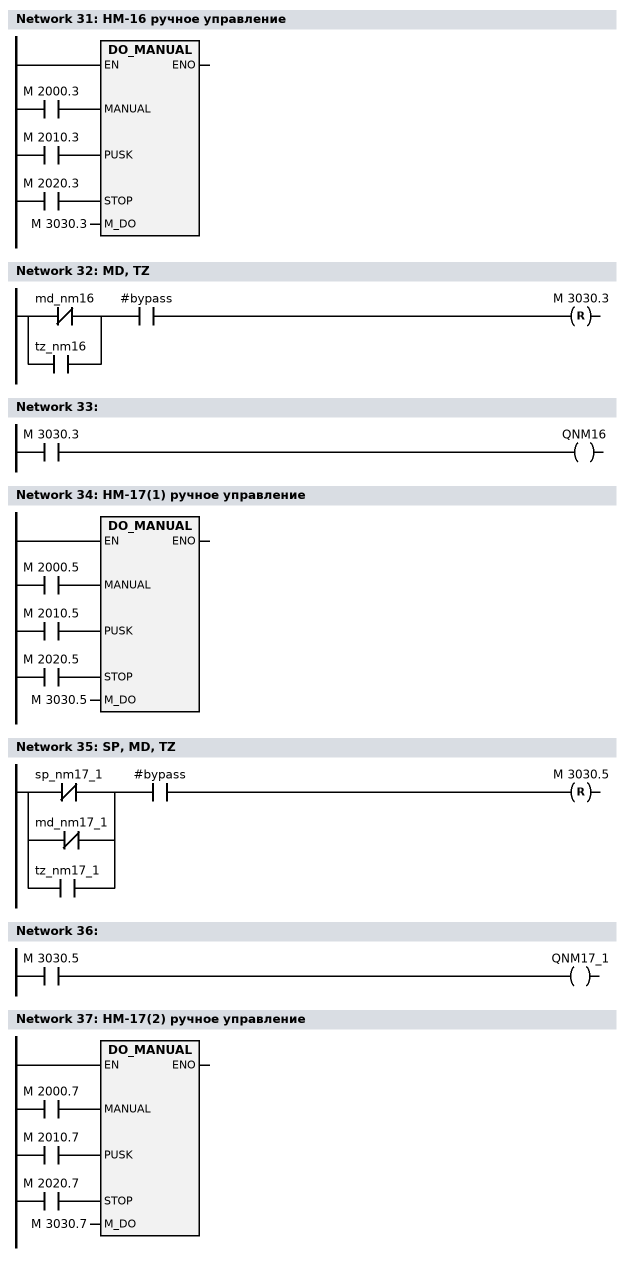
[picture p24: OB 1 networks 31-37]
NETWORK
TITLE = НМ-16 ручное управление
      A     M 2000.3;
      =     L 38.0;
      BLD   103;
      A     M 2010.3;
      =     L 38.1;
      BLD   103;
      A     M 2020.3;
      =     L 38.2;
      BLD   103;
      CALL  "DO_MANUAL" (
           MANUAL                   := L 38.0,
           PUSK                     := L 38.1,
           STOP                     := L 38.2,
           M_DO                     := M 3030.3);
      NOP   0;
NETWORK
TITLE = MD, TZ 
      A(;
      ON    "md_nm16";
      O     "tz_nm16";
      );
      A     #bypass;
      R     M 3030.3;
NETWORK
TITLE =
      A     M 3030.3;
      =     "QNM16";
NETWORK
TITLE = НМ-17(1) ручное управление
      A     M 2000.5;
      =     L 38.0;
      BLD   103;
      A     M 2010.5;
      =     L 38.1;
      BLD   103;
      A     M 2020.5;
      =     L 38.2;
      BLD   103;
      CALL  "DO_MANUAL" (
           MANUAL                   := L 38.0,
           PUSK                     := L 38.1,
           STOP                     := L 38.2,
           M_DO                     := M 3030.5);
      NOP   0;
NETWORK
TITLE = SP, MD, TZ 
      A(;
      ON    "sp_nm17_1";
      ON    "md_nm17_1";
      O     "tz_nm17_1";
      );
      A     #bypass;
      R     M 3030.5;
NETWORK
TITLE =
      A     M 3030.5;
      =     "QNM17_1";
NETWORK
TITLE = НМ-17(2) ручное управление
      A     M 2000.7;
      =     L 38.0;
      BLD   103;
      A     M 2010.7;
      =     L 38.1;
      BLD   103;
      A     M 2020.7;
      =     L 38.2;
      BLD   103;
      CALL  "DO_MANUAL" (
           MANUAL                   := L 38.0,
           PUSK                     := L 38.1,
           STOP                     := L 38.2,
           M_DO                     := M 3030.7);
      NOP   0;
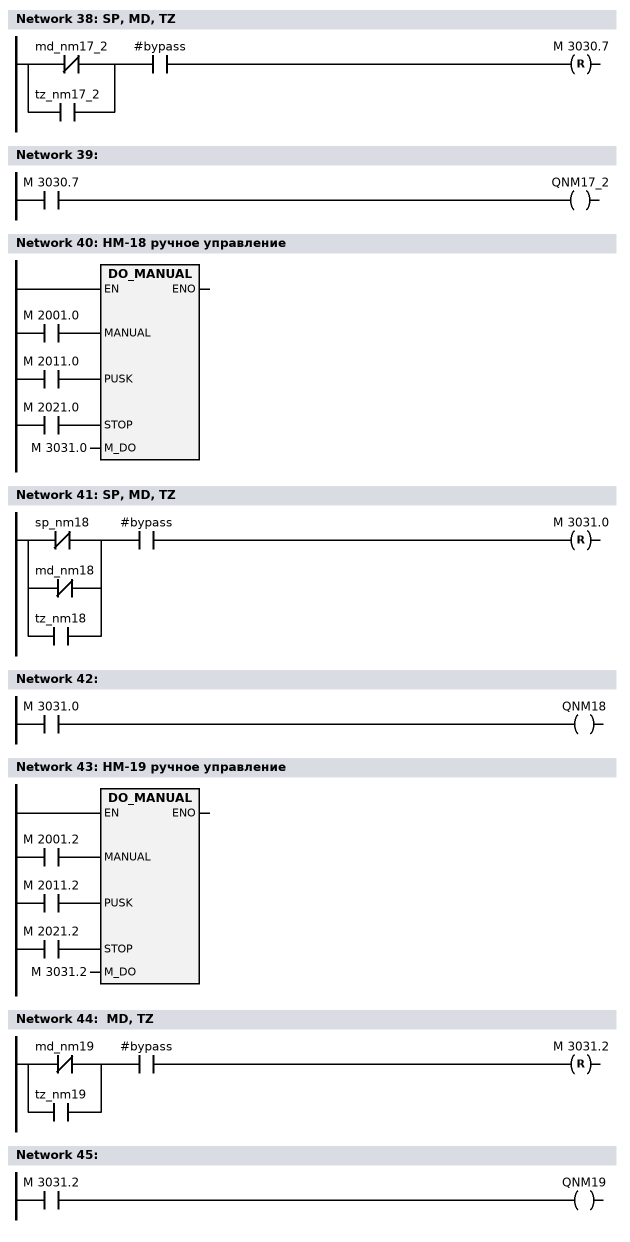
NETWORK
TITLE = SP, MD, TZ 
      A(;
      ON    "md_nm17_2";
      O     "tz_nm17_2";
      );
      A     #bypass;
      R     M 3030.7;
NETWORK
TITLE =
      A     M 3030.7;
      =     "QNM17_2";
NETWORK
TITLE = НМ-18 ручное управление
      A     M 2001.0;
      =     L 38.0;
      BLD   103;
      A     M 2011.0;
      =     L 38.1;
      BLD   103;
      A     M 2021.0;
      =     L 38.2;
      BLD   103;
      CALL  "DO_MANUAL" (
           MANUAL                   := L 38.0,
           PUSK                     := L 38.1,
           STOP                     := L 38.2,
           M_DO                     := M 3031.0);
      NOP   0;
NETWORK
TITLE = SP, MD, TZ 
      A(;
      ON    "sp_nm18";
      ON    "md_nm18";
      O     "tz_nm18";
      );
      A     #bypass;
      R     M 3031.0;
NETWORK
TITLE =
      A     M 3031.0;
      =     "QNM18";
NETWORK
TITLE = НМ-19 ручное управление
      A     M 2001.2;
      =     L 38.0;
      BLD   103;
      A     M 2011.2;
      =     L 38.1;
      BLD   103;
      A     M 2021.2;
      =     L 38.2;
      BLD   103;
      CALL  "DO_MANUAL" (
           MANUAL                   := L 38.0,
           PUSK                     := L 38.1,
           STOP                     := L 38.2,
           M_DO                     := M 3031.2);
      NOP   0;
NETWORK
TITLE =  MD, TZ 
      A(;
      ON    "md_nm19";
      O     "tz_nm19";
      );
      A     #bypass;
      R     M 3031.2;
NETWORK
TITLE =
      A     M 3031.2;
      =     "QNM19";
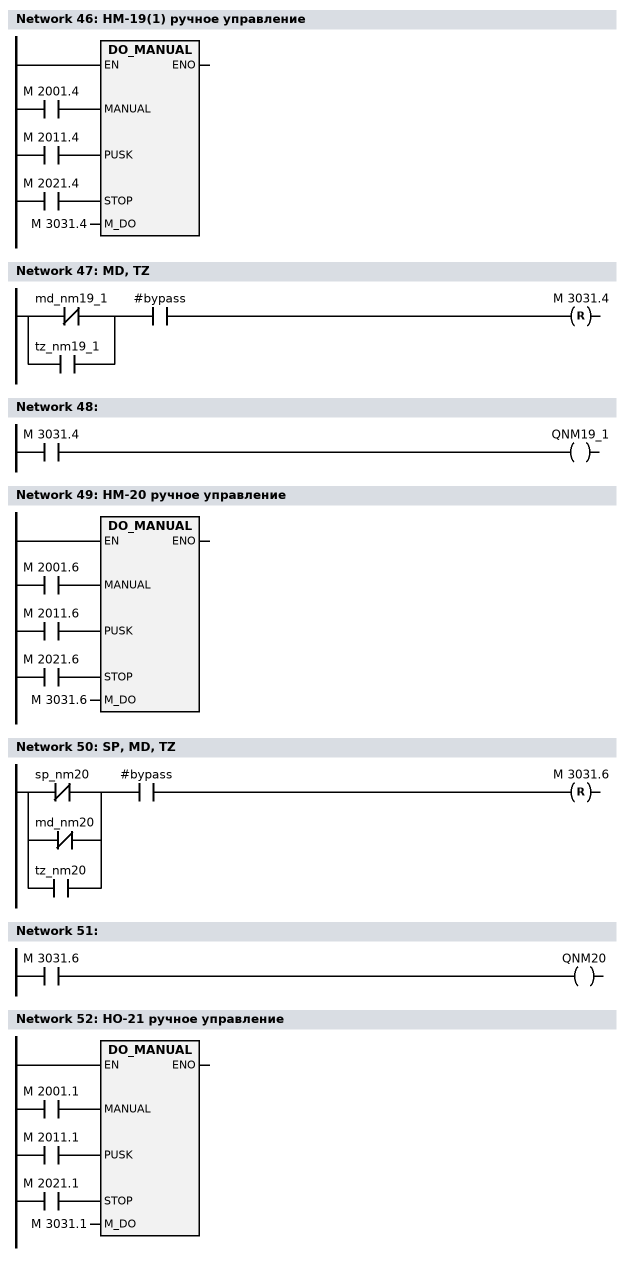
NETWORK
TITLE = НМ-19(1) ручное управление
      A     M 2001.4;
      =     L 38.0;
      BLD   103;
      A     M 2011.4;
      =     L 38.1;
      BLD   103;
      A     M 2021.4;
      =     L 38.2;
      BLD   103;
      CALL  "DO_MANUAL" (
           MANUAL                   := L 38.0,
           PUSK                     := L 38.1,
           STOP                     := L 38.2,
           M_DO                     := M 3031.4);
      NOP   0;
NETWORK
TITLE = MD, TZ 
      A(;
      ON    "md_nm19_1";
      O     "tz_nm19_1";
      );
      A     #bypass;
      R     M 3031.4;
NETWORK
TITLE =
      A     M 3031.4;
      =     "QNM19_1";
NETWORK
TITLE = НМ-20 ручное управление
      A     M 2001.6;
      =     L 38.0;
      BLD   103;
      A     M 2011.6;
      =     L 38.1;
      BLD   103;
      A     M 2021.6;
      =     L 38.2;
      BLD   103;
      CALL  "DO_MANUAL" (
           MANUAL                   := L 38.0,
           PUSK                     := L 38.1,
           STOP                     := L 38.2,
           M_DO                     := M 3031.6);
      NOP   0;
NETWORK
TITLE = SP, MD, TZ 
      A(;
      ON    "sp_nm20";
      ON    "md_nm20";
      O     "tz_nm20";
      );
      A     #bypass;
      R     M 3031.6;
NETWORK
TITLE =
      A     M 3031.6;
      =     "QNM20";
NETWORK
TITLE = НО-21 ручное управление
      A     M 2001.1;
      =     L 38.0;
      BLD   103;
      A     M 2011.1;
      =     L 38.1;
      BLD   103;
      A     M 2021.1;
      =     L 38.2;
      BLD   103;
      CALL  "DO_MANUAL" (
           MANUAL                   := L 38.0,
           PUSK                     := L 38.1,
           STOP                     := L 38.2,
           M_DO                     := M 3031.1);
      NOP   0;
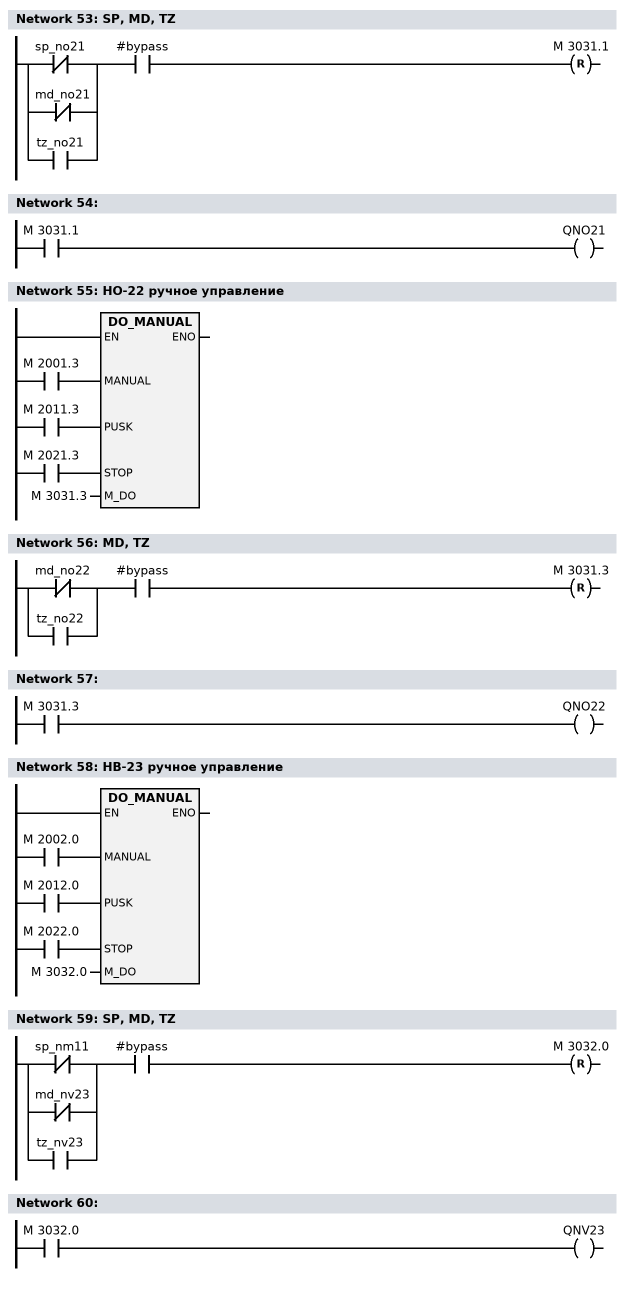
NETWORK
TITLE = SP, MD, TZ 
      A(;
      ON    "sp_no21";
      ON    "md_no21";
      O     "tz_no21";
      );
      A     #bypass;
      R     M 3031.1;
NETWORK
TITLE =
      A     M 3031.1;
      =     "QNO21";
NETWORK
TITLE = НО-22 ручное управление
      A     M 2001.3;
      =     L 38.0;
      BLD   103;
      A     M 2011.3;
      =     L 38.1;
      BLD   103;
      A     M 2021.3;
      =     L 38.2;
      BLD   103;
      CALL  "DO_MANUAL" (
           MANUAL                   := L 38.0,
           PUSK                     := L 38.1,
           STOP                     := L 38.2,
           M_DO                     := M 3031.3);
      NOP   0;
NETWORK
TITLE = MD, TZ 
      A(;
      ON    "md_no22";
      O     "tz_no22";
      );
      A     #bypass;
      R     M 3031.3;
NETWORK
TITLE =
      A     M 3031.3;
      =     "QNO22";
NETWORK
TITLE = НВ-23 ручное управление
      A     M 2002.0;
      =     L 38.0;
      BLD   103;
      A     M 2012.0;
      =     L 38.1;
      BLD   103;
      A     M 2022.0;
      =     L 38.2;
      BLD   103;
      CALL  "DO_MANUAL" (
           MANUAL                   := L 38.0,
           PUSK                     := L 38.1,
           STOP                     := L 38.2,
           M_DO                     := M 3032.0);
      NOP   0;
NETWORK
TITLE = SP, MD, TZ 
      A(;
      ON    "sp_nm11";
      ON    "md_nv23";
      O     "tz_nv23";
      );
      A     #bypass;
      R     M 3032.0;
NETWORK
TITLE =
      A     M 3032.0;
      =     "QNV23";
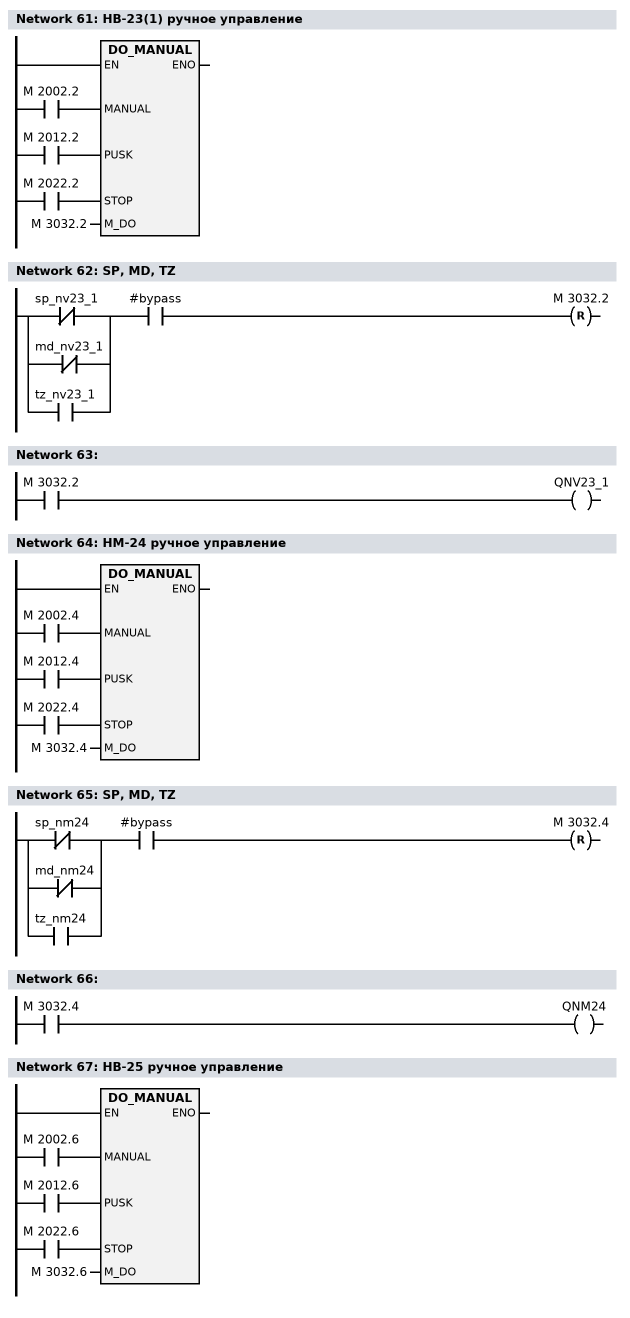
NETWORK
TITLE = НВ-23(1) ручное управление
      A     M 2002.2;
      =     L 38.0;
      BLD   103;
      A     M 2012.2;
      =     L 38.1;
      BLD   103;
      A     M 2022.2;
      =     L 38.2;
      BLD   103;
      CALL  "DO_MANUAL" (
           MANUAL                   := L 38.0,
           PUSK                     := L 38.1,
           STOP                     := L 38.2,
           M_DO                     := M 3032.2);
      NOP   0;
NETWORK
TITLE = SP, MD, TZ 
      A(;
      ON    "sp_nv23_1";
      ON    "md_nv23_1";
      O     "tz_nv23_1";
      );
      A     #bypass;
      R     M 3032.2;
NETWORK
TITLE =
      A     M 3032.2;
      =     "QNV23_1";
NETWORK
TITLE = НМ-24 ручное управление
      A     M 2002.4;
      =     L 38.0;
      BLD   103;
      A     M 2012.4;
      =     L 38.1;
      BLD   103;
      A     M 2022.4;
      =     L 38.2;
      BLD   103;
      CALL  "DO_MANUAL" (
           MANUAL                   := L 38.0,
           PUSK                     := L 38.1,
           STOP                     := L 38.2,
           M_DO                     := M 3032.4);
      NOP   0;
NETWORK
TITLE = SP, MD, TZ 
      A(;
      ON    "sp_nm24";
      ON    "md_nm24";
      O     "tz_nm24";
      );
      A     #bypass;
      R     M 3032.4;
NETWORK
TITLE =
      A     M 3032.4;
      =     "QNM24";
NETWORK
TITLE = НВ-25 ручное управление
      A     M 2002.6;
      =     L 38.0;
      BLD   103;
      A     M 2012.6;
      =     L 38.1;
      BLD   103;
      A     M 2022.6;
      =     L 38.2;
      BLD   103;
      CALL  "DO_MANUAL" (
           MANUAL                   := L 38.0,
           PUSK                     := L 38.1,
           STOP                     := L 38.2,
           M_DO                     := M 3032.6);
      NOP   0;
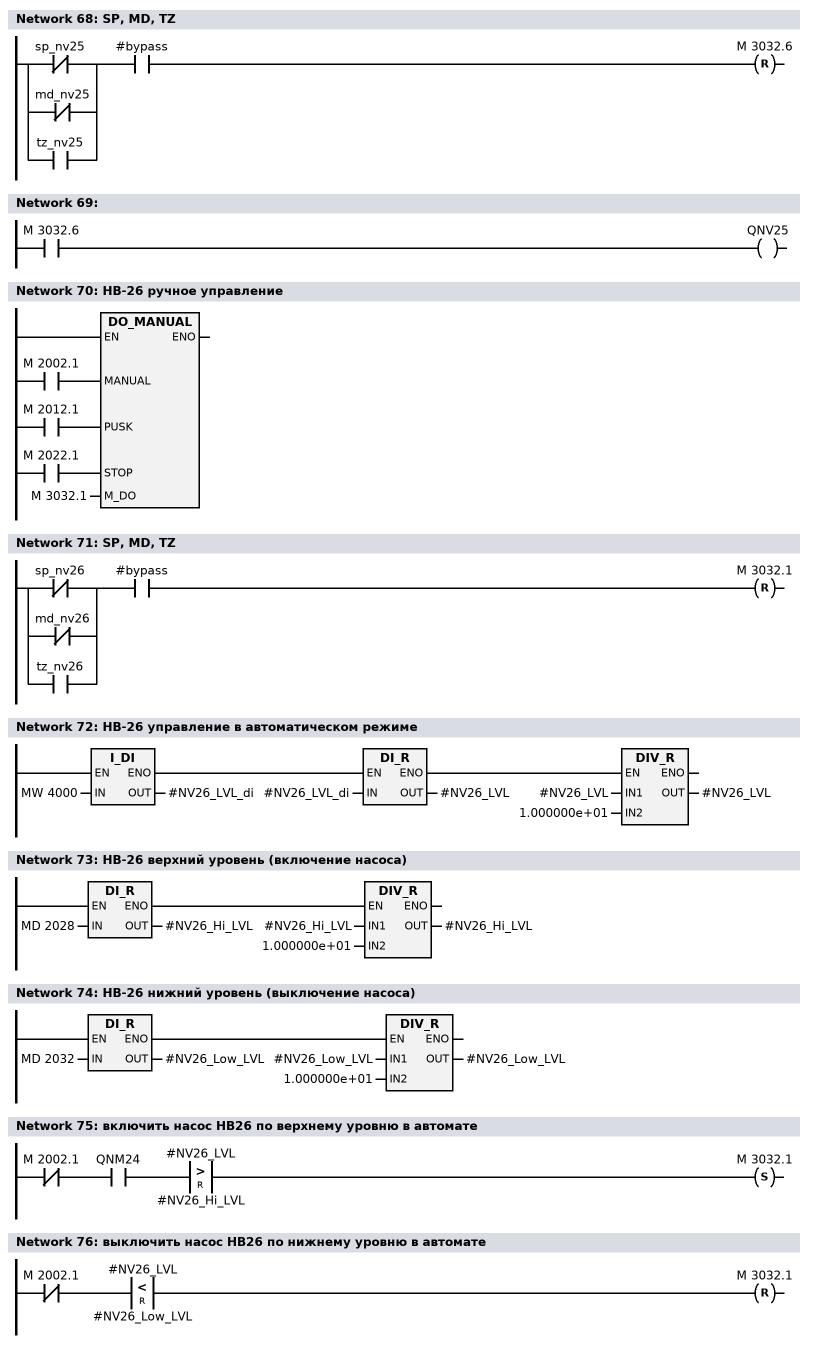
NETWORK
TITLE = SP, MD, TZ 
      A(;
      ON    "sp_nv25";
      ON    "md_nv25";
      O     "tz_nv25";
      );
      A     #bypass;
      R     M 3032.6;
NETWORK
TITLE =
      A     M 3032.6;
      =     "QNV25";
NETWORK
TITLE = НВ-26 ручное управление
      A     M 2002.1;
      =     L 38.0;
      BLD   103;
      A     M 2012.1;
      =     L 38.1;
      BLD   103;
      A     M 2022.1;
      =     L 38.2;
      BLD   103;
      CALL  "DO_MANUAL" (
           MANUAL                   := L 38.0,
           PUSK                     := L 38.1,
           STOP                     := L 38.2,
           M_DO                     := M 3032.1);
      NOP   0;
NETWORK
TITLE = SP, MD, TZ 
      A(;
      ON    "sp_nv26";
      ON    "md_nv26";
      O     "tz_nv26";
      );
      A     #bypass;
      R     M 3032.1;
NETWORK
TITLE = НВ-26 управление в автоматическом режиме
//Уровень в баке крофты
      A(;
      A(;
      L     MW 4000;
      ITD;
      T     #NV26_LVL_di;
      SET;
      SAVE;
      CLR;
      A     BR;
      );
      JNB   _001;
      L     #NV26_LVL_di;
      DTR;
      T     #NV26_LVL;
      SET;
      SAVE;
      CLR;
_001: A     BR;
      );
      JNB   _002;
      L     #NV26_LVL;
      L     1.000000e+01;
      /R;
      T     #NV26_LVL;
_002: NOP   0;
NETWORK
TITLE = НВ-26 верхний уровень (включение насоса)
      A(;
      L     MD 2028;
      DTR;
      T     #NV26_Hi_LVL;
      SET;
      SAVE;
      CLR;
      A     BR;
      );
      JNB   _003;
      L     #NV26_Hi_LVL;
      L     1.000000e+01;
      /R;
      T     #NV26_Hi_LVL;
_003: NOP   0;
NETWORK
TITLE = НВ-26 нижний уровень (выключение насоса)
      A(;
      L     MD 2032;
      DTR;
      T     #NV26_Low_LVL;
      SET;
      SAVE;
      CLR;
      A     BR;
      );
      JNB   _004;
      L     #NV26_Low_LVL;
      L     1.000000e+01;
      /R;
      T     #NV26_Low_LVL;
_004: NOP   0;
NETWORK
TITLE = включить насос НВ26 по верхнему уровню в автомате
      AN    M 2002.1;
      A     "QNM24";
      A(;
      L     #NV26_LVL;
      L     #NV26_Hi_LVL;
      >R;
      );
      S     M 3032.1;
NETWORK
TITLE = выключить насос НВ26 по нижнему уровню в автомате
      AN    M 2002.1;
      A(;
      L     #NV26_LVL;
      L     #NV26_Low_LVL;
      <R;
      );
      R     M 3032.1;
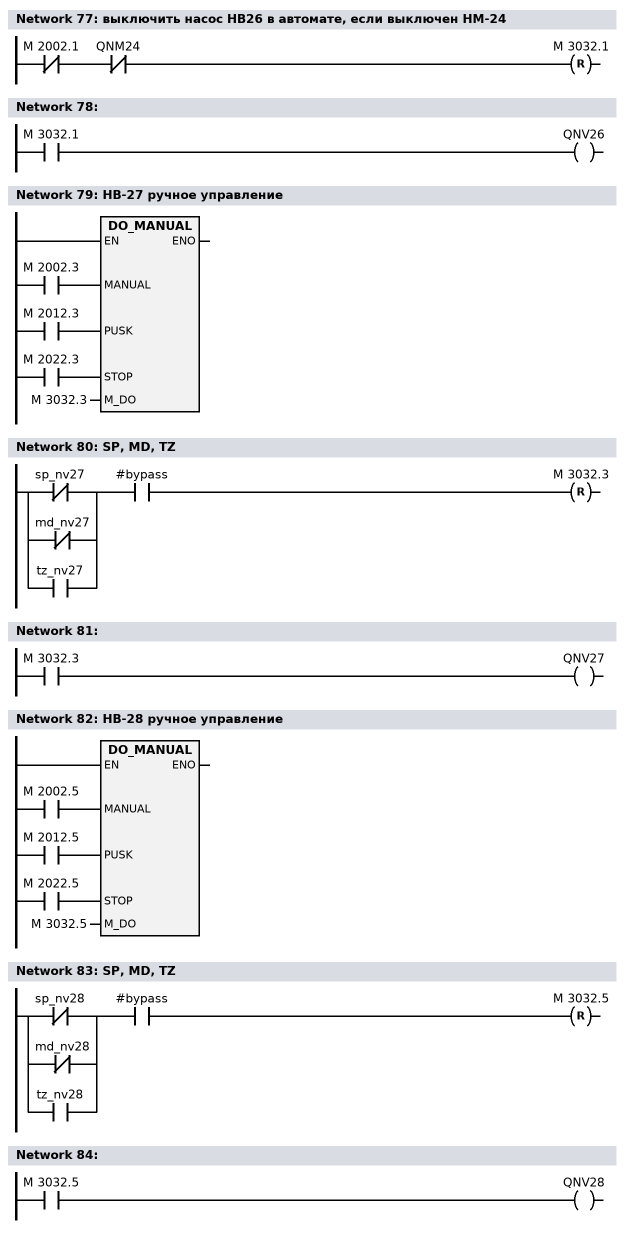
NETWORK
TITLE = выключить насос НВ26 в автомате, если выключен НМ-24 
      AN    M 2002.1;
      AN    "QNM24";
      R     M 3032.1;
NETWORK
TITLE =
      A     M 3032.1;
      =     "QNV26";
NETWORK
TITLE = НВ-27 ручное управление
//******************************************************************************
      A     M 2002.3;
      =     L 38.0;
      BLD   103;
      A     M 2012.3;
      =     L 38.1;
      BLD   103;
      A     M 2022.3;
      =     L 38.2;
      BLD   103;
      CALL  "DO_MANUAL" (
           MANUAL                   := L 38.0,
           PUSK                     := L 38.1,
           STOP                     := L 38.2,
           M_DO                     := M 3032.3);
      NOP   0;
NETWORK
TITLE = SP, MD, TZ 
      A(;
      ON    "sp_nv27";
      ON    "md_nv27";
      O     "tz_nv27";
      );
      A     #bypass;
      R     M 3032.3;
NETWORK
TITLE =
      A     M 3032.3;
      =     "QNV27";
NETWORK
TITLE = НВ-28 ручное управление
      A     M 2002.5;
      =     L 38.0;
      BLD   103;
      A     M 2012.5;
      =     L 38.1;
      BLD   103;
      A     M 2022.5;
      =     L 38.2;
      BLD   103;
      CALL  "DO_MANUAL" (
           MANUAL                   := L 38.0,
           PUSK                     := L 38.1,
           STOP                     := L 38.2,
           M_DO                     := M 3032.5);
      NOP   0;
NETWORK
TITLE = SP, MD, TZ 
      A(;
      ON    "sp_nv28";
      ON    "md_nv28";
      O     "tz_nv28";
      );
      A     #bypass;
      R     M 3032.5;
NETWORK
TITLE =
      A     M 3032.5;
      =     "QNV28";
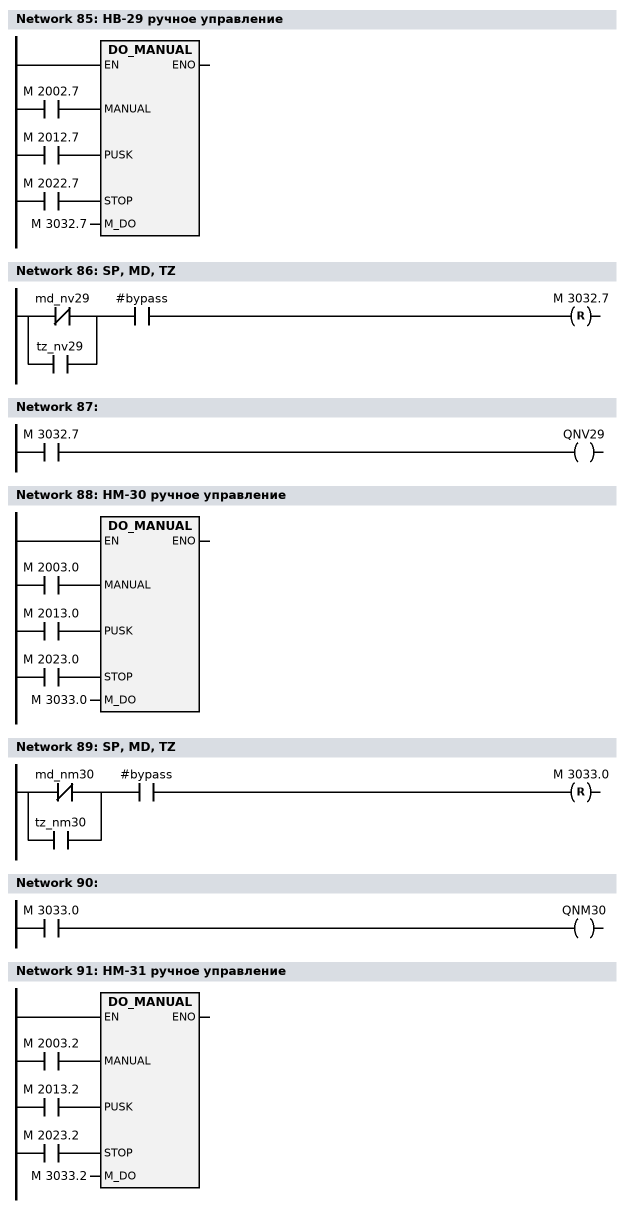
NETWORK
TITLE = НВ-29 ручное управление
      A     M 2002.7;
      =     L 38.0;
      BLD   103;
      A     M 2012.7;
      =     L 38.1;
      BLD   103;
      A     M 2022.7;
      =     L 38.2;
      BLD   103;
      CALL  "DO_MANUAL" (
           MANUAL                   := L 38.0,
           PUSK                     := L 38.1,
           STOP                     := L 38.2,
           M_DO                     := M 3032.7);
      NOP   0;
NETWORK
TITLE = SP, MD, TZ 
      A(;
      ON    "md_nv29";
      O     "tz_nv29";
      );
      A     #bypass;
      R     M 3032.7;
NETWORK
TITLE =
      A     M 3032.7;
      =     "QNV29";
NETWORK
TITLE = НМ-30 ручное управление
      A     M 2003.0;
      =     L 38.0;
      BLD   103;
      A     M 2013.0;
      =     L 38.1;
      BLD   103;
      A     M 2023.0;
      =     L 38.2;
      BLD   103;
      CALL  "DO_MANUAL" (
           MANUAL                   := L 38.0,
           PUSK                     := L 38.1,
           STOP                     := L 38.2,
           M_DO                     := M 3033.0);
      NOP   0;
NETWORK
TITLE = SP, MD, TZ 
      A(;
      ON    "md_nm30";
      O     "tz_nm30";
      );
      A     #bypass;
      R     M 3033.0;
NETWORK
TITLE =
      A     M 3033.0;
      =     "QNM30";
NETWORK
TITLE = НМ-31 ручное управление
      A     M 2003.2;
      =     L 38.0;
      BLD   103;
      A     M 2013.2;
      =     L 38.1;
      BLD   103;
      A     M 2023.2;
      =     L 38.2;
      BLD   103;
      CALL  "DO_MANUAL" (
           MANUAL                   := L 38.0,
           PUSK                     := L 38.1,
           STOP                     := L 38.2,
           M_DO                     := M 3033.2);
      NOP   0;
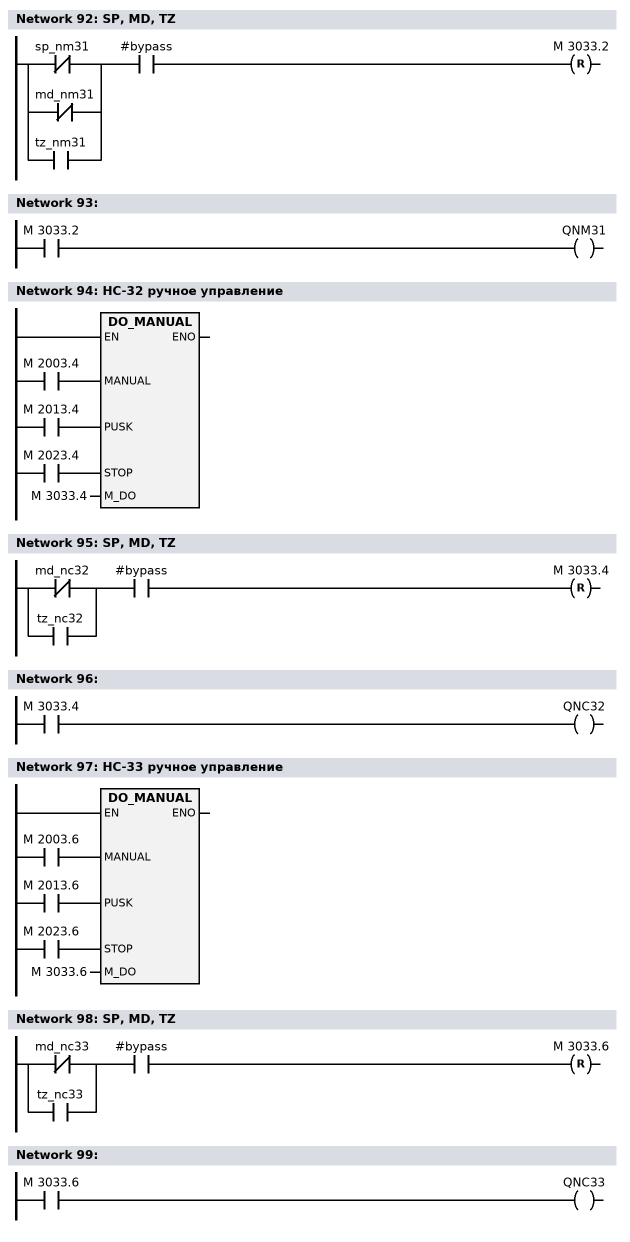
NETWORK
TITLE = SP, MD, TZ 
      A(;
      ON    "sp_nm31";
      ON    "md_nm31";
      O     "tz_nm31";
      );
      A     #bypass;
      R     M 3033.2;
NETWORK
TITLE =
      A     M 3033.2;
      =     "QNM31";
NETWORK
TITLE = НС-32 ручное управление
      A     M 2003.4;
      =     L 38.0;
      BLD   103;
      A     M 2013.4;
      =     L 38.1;
      BLD   103;
      A     M 2023.4;
      =     L 38.2;
      BLD   103;
      CALL  "DO_MANUAL" (
           MANUAL                   := L 38.0,
           PUSK                     := L 38.1,
           STOP                     := L 38.2,
           M_DO                     := M 3033.4);
      NOP   0;
NETWORK
TITLE = SP, MD, TZ 
      A(;
      ON    "md_nc32";
      O     "tz_nc32";
      );
      A     #bypass;
      R     M 3033.4;
NETWORK
TITLE =
      A     M 3033.4;
      =     "QNC32";
NETWORK
TITLE = НС-33 ручное управление
      A     M 2003.6;
      =     L 38.0;
      BLD   103;
      A     M 2013.6;
      =     L 38.1;
      BLD   103;
      A     M 2023.6;
      =     L 38.2;
      BLD   103;
      CALL  "DO_MANUAL" (
           MANUAL                   := L 38.0,
           PUSK                     := L 38.1,
           STOP                     := L 38.2,
           M_DO                     := M 3033.6);
      NOP   0;
NETWORK
TITLE = SP, MD, TZ 
      A(;
      ON    "md_nc33";
      O     "tz_nc33";
      );
      A     #bypass;
      R     M 3033.6;
NETWORK
TITLE =
      A     M 3033.6;
      =     "QNC33";
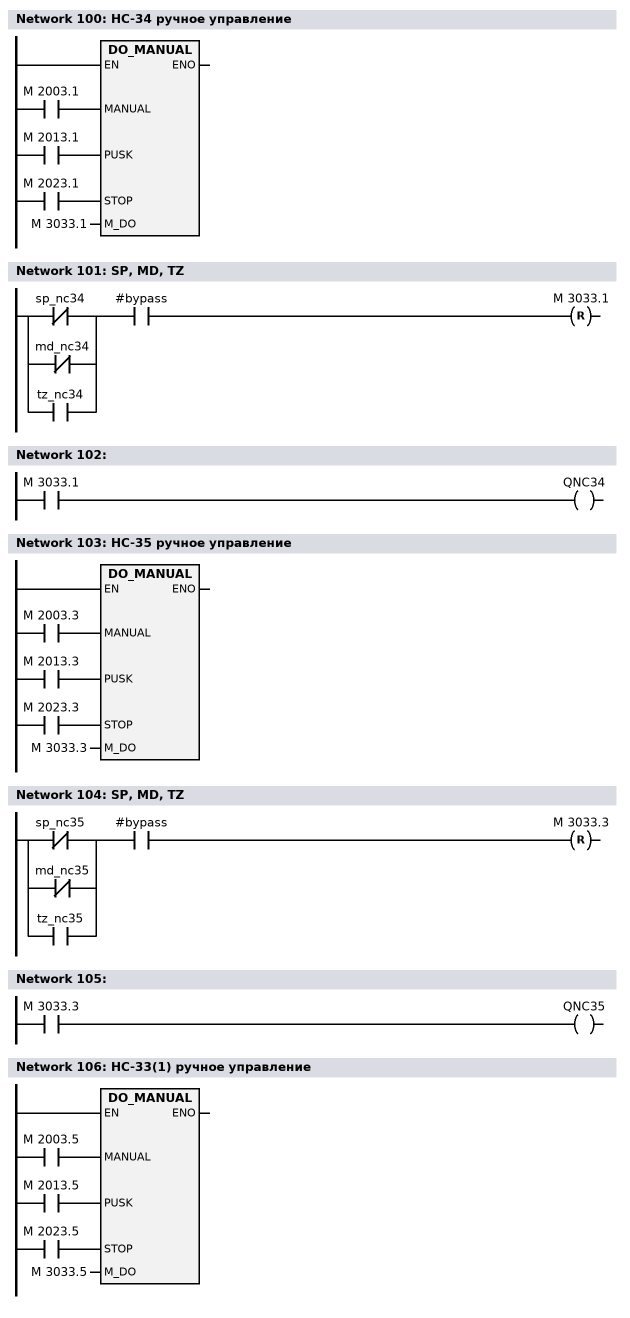
NETWORK
TITLE = НС-34 ручное управление
      A     M 2003.1;
      =     L 38.0;
      BLD   103;
      A     M 2013.1;
      =     L 38.1;
      BLD   103;
      A     M 2023.1;
      =     L 38.2;
      BLD   103;
      CALL  "DO_MANUAL" (
           MANUAL                   := L 38.0,
           PUSK                     := L 38.1,
           STOP                     := L 38.2,
           M_DO                     := M 3033.1);
      NOP   0;
NETWORK
TITLE = SP, MD, TZ 
      A(;
      ON    "sp_nc34";
      ON    "md_nc34";
      O     "tz_nc34";
      );
      A     #bypass;
      R     M 3033.1;
NETWORK
TITLE =
      A     M 3033.1;
      =     "QNC34";
NETWORK
TITLE = НС-35 ручное управление
      A     M 2003.3;
      =     L 38.0;
      BLD   103;
      A     M 2013.3;
      =     L 38.1;
      BLD   103;
      A     M 2023.3;
      =     L 38.2;
      BLD   103;
      CALL  "DO_MANUAL" (
           MANUAL                   := L 38.0,
           PUSK                     := L 38.1,
           STOP                     := L 38.2,
           M_DO                     := M 3033.3);
      NOP   0;
NETWORK
TITLE = SP, MD, TZ 
      A(;
      ON    "sp_nc35";
      ON    "md_nc35";
      O     "tz_nc35";
      );
      A     #bypass;
      R     M 3033.3;
NETWORK
TITLE =
      A     M 3033.3;
      =     "QNC35";
NETWORK
TITLE = НС-33(1) ручное управление
      A     M 2003.5;
      =     L 38.0;
      BLD   103;
      A     M 2013.5;
      =     L 38.1;
      BLD   103;
      A     M 2023.5;
      =     L 38.2;
      BLD   103;
      CALL  "DO_MANUAL" (
           MANUAL                   := L 38.0,
           PUSK                     := L 38.1,
           STOP                     := L 38.2,
           M_DO                     := M 3033.5);
      NOP   0;
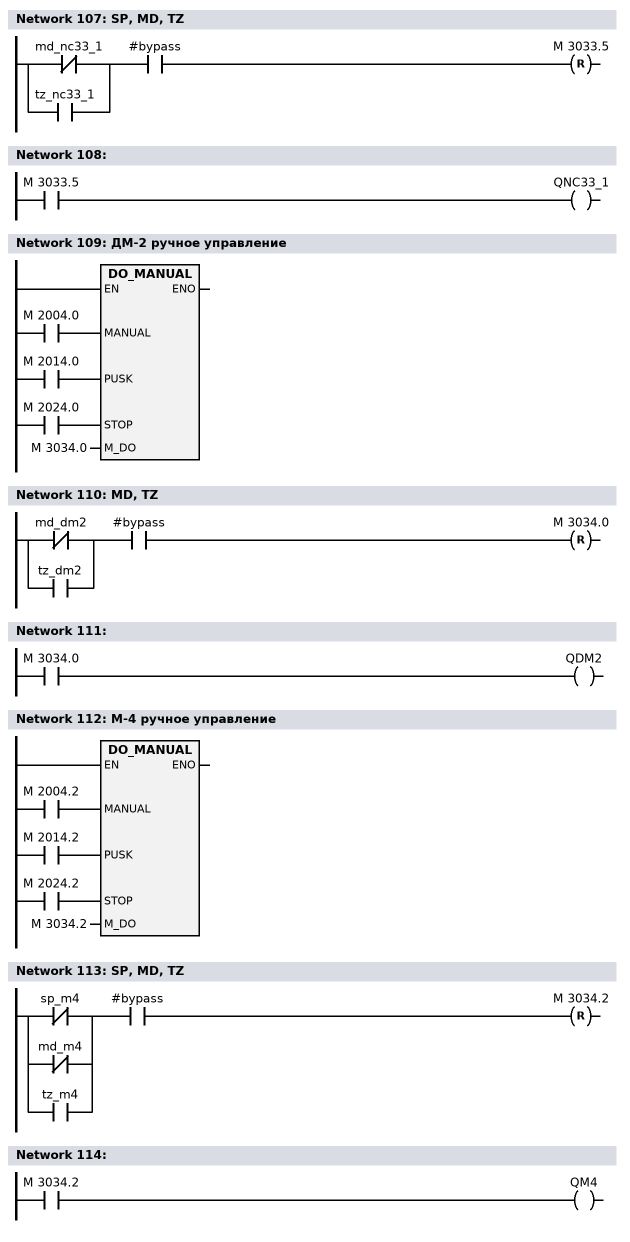
NETWORK
TITLE = SP, MD, TZ 
      A(;
      ON    "md_nc33_1";
      O     "tz_nc33_1";
      );
      A     #bypass;
      R     M 3033.5;
NETWORK
TITLE =
      A     M 3033.5;
      =     "QNC33_1";
NETWORK
TITLE = ДМ-2 ручное управление
      A     M 2004.0;
      =     L 38.0;
      BLD   103;
      A     M 2014.0;
      =     L 38.1;
      BLD   103;
      A     M 2024.0;
      =     L 38.2;
      BLD   103;
      CALL  "DO_MANUAL" (
           MANUAL                   := L 38.0,
           PUSK                     := L 38.1,
           STOP                     := L 38.2,
           M_DO                     := M 3034.0);
      NOP   0;
NETWORK
TITLE = MD, TZ 
      A(;
      ON    "md_dm2";
      O     "tz_dm2";
      );
      A     #bypass;
      R     M 3034.0;
NETWORK
TITLE =
      A     M 3034.0;
      =     "QDM2";
NETWORK
TITLE = М-4 ручное управление
      A     M 2004.2;
      =     L 38.0;
      BLD   103;
      A     M 2014.2;
      =     L 38.1;
      BLD   103;
      A     M 2024.2;
      =     L 38.2;
      BLD   103;
      CALL  "DO_MANUAL" (
           MANUAL                   := L 38.0,
           PUSK                     := L 38.1,
           STOP                     := L 38.2,
           M_DO                     := M 3034.2);
      NOP   0;
NETWORK
TITLE = SP, MD, TZ 
      A(;
      ON    "sp_m4";
      ON    "md_m4";
      O     "tz_m4";
      );
      A     #bypass;
      R     M 3034.2;
NETWORK
TITLE =
      A     M 3034.2;
      =     "QM4";
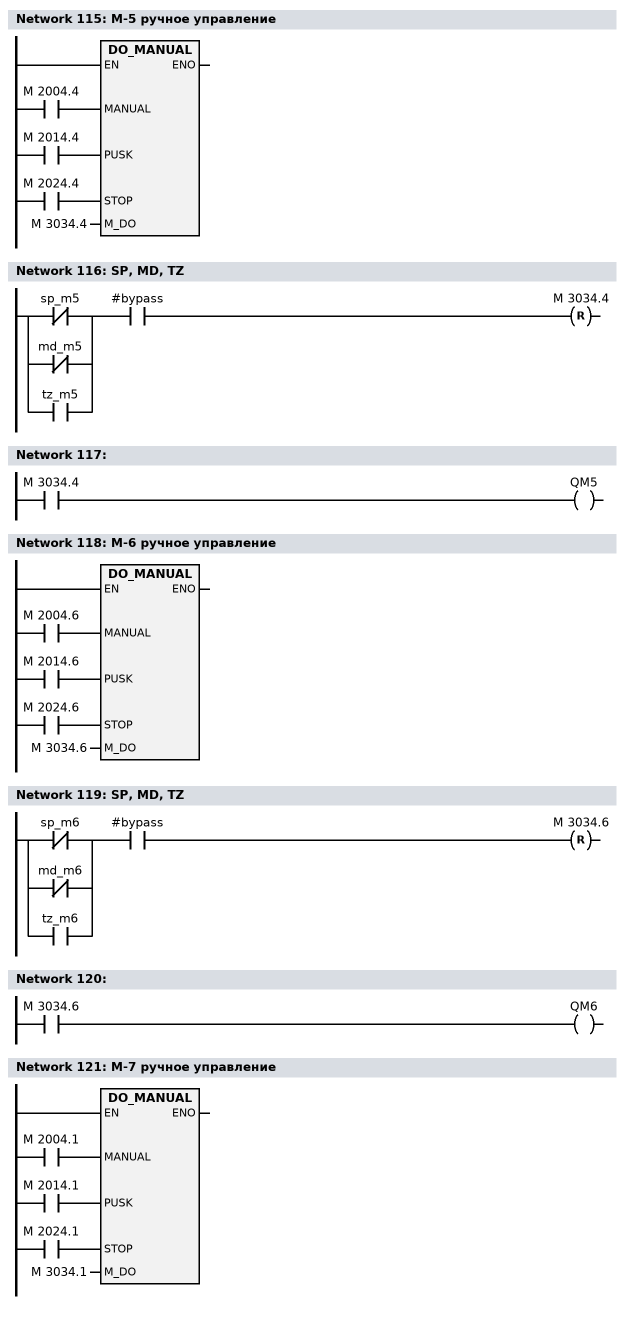
NETWORK
TITLE = М-5 ручное управление
      A     M 2004.4;
      =     L 38.0;
      BLD   103;
      A     M 2014.4;
      =     L 38.1;
      BLD   103;
      A     M 2024.4;
      =     L 38.2;
      BLD   103;
      CALL  "DO_MANUAL" (
           MANUAL                   := L 38.0,
           PUSK                     := L 38.1,
           STOP                     := L 38.2,
           M_DO                     := M 3034.4);
      NOP   0;
NETWORK
TITLE = SP, MD, TZ 
      A(;
      ON    "sp_m5";
      ON    "md_m5";
      O     "tz_m5";
      );
      A     #bypass;
      R     M 3034.4;
NETWORK
TITLE =
      A     M 3034.4;
      =     "QM5";
NETWORK
TITLE = М-6 ручное управление
      A     M 2004.6;
      =     L 38.0;
      BLD   103;
      A     M 2014.6;
      =     L 38.1;
      BLD   103;
      A     M 2024.6;
      =     L 38.2;
      BLD   103;
      CALL  "DO_MANUAL" (
           MANUAL                   := L 38.0,
           PUSK                     := L 38.1,
           STOP                     := L 38.2,
           M_DO                     := M 3034.6);
      NOP   0;
NETWORK
TITLE = SP, MD, TZ 
      A(;
      ON    "sp_m6";
      ON    "md_m6";
      O     "tz_m6";
      );
      A     #bypass;
      R     M 3034.6;
NETWORK
TITLE =
      A     M 3034.6;
      =     "QM6";
NETWORK
TITLE = М-7 ручное управление
      A     M 2004.1;
      =     L 38.0;
      BLD   103;
      A     M 2014.1;
      =     L 38.1;
      BLD   103;
      A     M 2024.1;
      =     L 38.2;
      BLD   103;
      CALL  "DO_MANUAL" (
           MANUAL                   := L 38.0,
           PUSK                     := L 38.1,
           STOP                     := L 38.2,
           M_DO                     := M 3034.1);
      NOP   0;
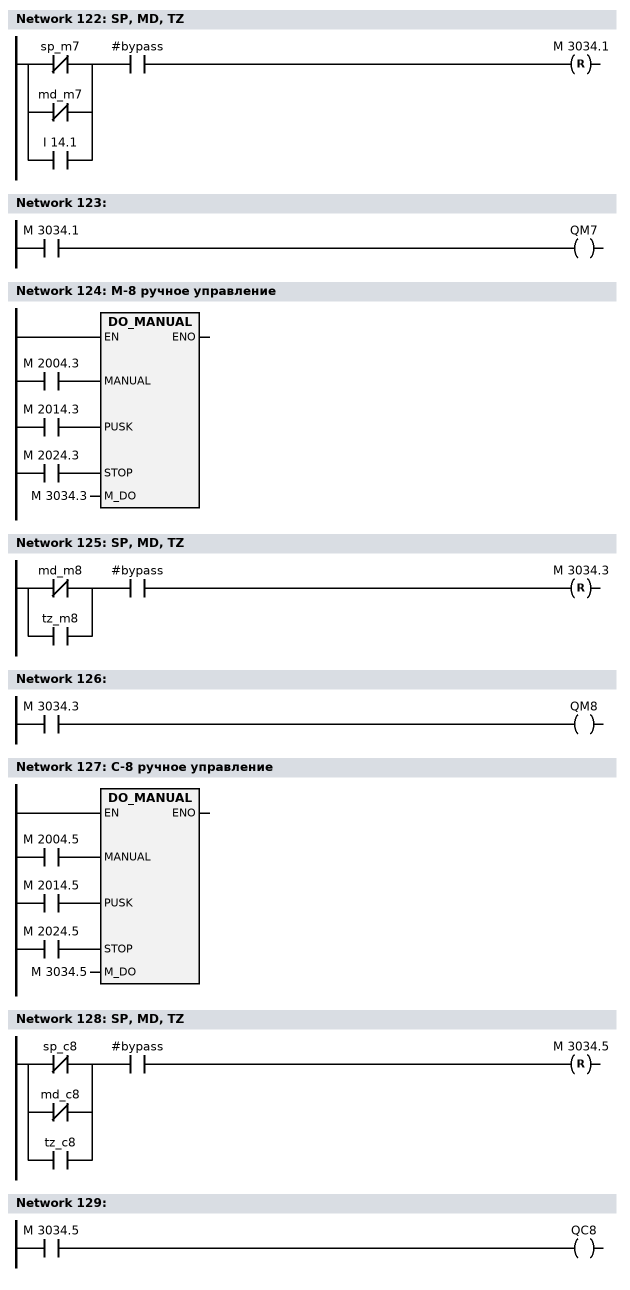
NETWORK
TITLE = SP, MD, TZ 
      A(;
      ON    "sp_m7";
      ON    "md_m7";
      O     I 14.1;
      );
      A     #bypass;
      R     M 3034.1;
NETWORK
TITLE =
      A     M 3034.1;
      =     "QM7";
NETWORK
TITLE = М-8 ручное управление
      A     M 2004.3;
      =     L 38.0;
      BLD   103;
      A     M 2014.3;
      =     L 38.1;
      BLD   103;
      A     M 2024.3;
      =     L 38.2;
      BLD   103;
      CALL  "DO_MANUAL" (
           MANUAL                   := L 38.0,
           PUSK                     := L 38.1,
           STOP                     := L 38.2,
           M_DO                     := M 3034.3);
      NOP   0;
NETWORK
TITLE = SP, MD, TZ 
      A(;
      ON    "md_m8";
      O     "tz_m8";
      );
      A     #bypass;
      R     M 3034.3;
NETWORK
TITLE =
      A     M 3034.3;
      =     "QM8";
NETWORK
TITLE = C-8 ручное управление
      A     M 2004.5;
      =     L 38.0;
      BLD   103;
      A     M 2014.5;
      =     L 38.1;
      BLD   103;
      A     M 2024.5;
      =     L 38.2;
      BLD   103;
      CALL  "DO_MANUAL" (
           MANUAL                   := L 38.0,
           PUSK                     := L 38.1,
           STOP                     := L 38.2,
           M_DO                     := M 3034.5);
      NOP   0;
NETWORK
TITLE = SP, MD, TZ 
      A(;
      ON    "sp_c8";
      ON    "md_c8";
      O     "tz_c8";
      );
      A     #bypass;
      R     M 3034.5;
NETWORK
TITLE =
      A     M 3034.5;
      =     "QC8";
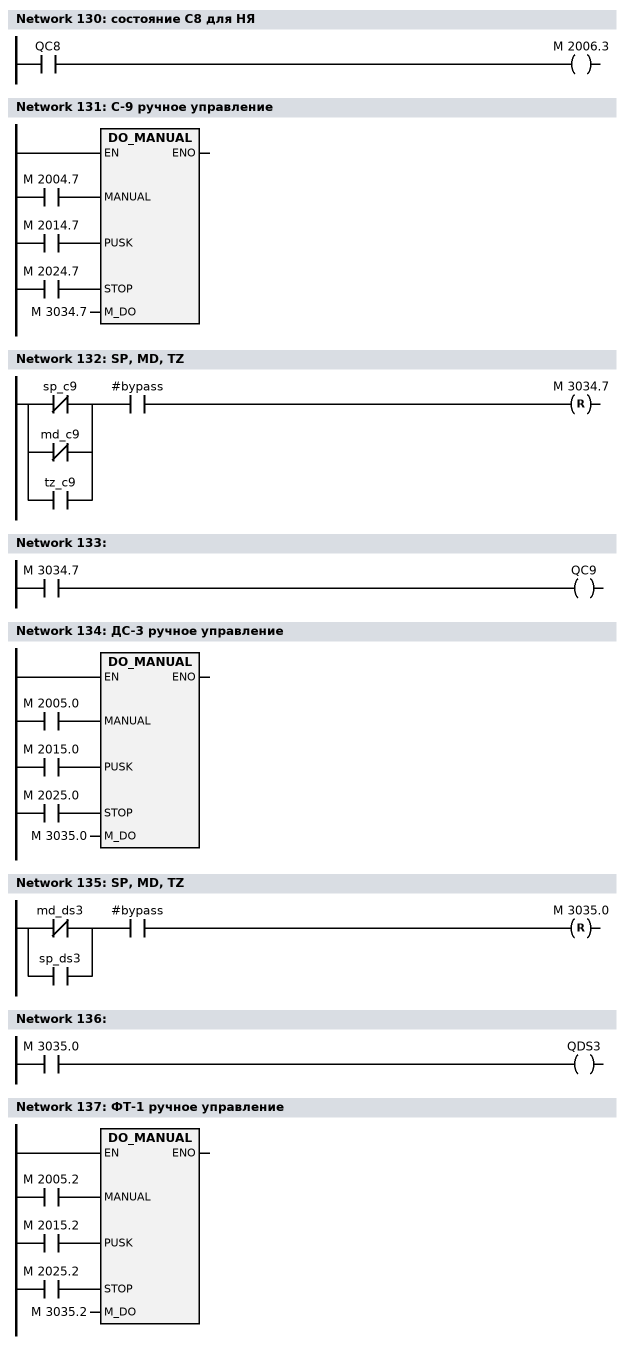
NETWORK
TITLE = состояние С8 для НЯ
      A     "QC8";
      =     M 2006.3;
NETWORK
TITLE = C-9 ручное управление
      A     M 2004.7;
      =     L 38.0;
      BLD   103;
      A     M 2014.7;
      =     L 38.1;
      BLD   103;
      A     M 2024.7;
      =     L 38.2;
      BLD   103;
      CALL  "DO_MANUAL" (
           MANUAL                   := L 38.0,
           PUSK                     := L 38.1,
           STOP                     := L 38.2,
           M_DO                     := M 3034.7);
      NOP   0;
NETWORK
TITLE = SP, MD, TZ 
      A(;
      ON    "sp_c9";
      ON    "md_c9";
      O     "tz_c9";
      );
      A     #bypass;
      R     M 3034.7;
NETWORK
TITLE =
      A     M 3034.7;
      =     "QC9";
NETWORK
TITLE = ДС-3 ручное управление
      A     M 2005.0;
      =     L 38.0;
      BLD   103;
      A     M 2015.0;
      =     L 38.1;
      BLD   103;
      A     M 2025.0;
      =     L 38.2;
      BLD   103;
      CALL  "DO_MANUAL" (
           MANUAL                   := L 38.0,
           PUSK                     := L 38.1,
           STOP                     := L 38.2,
           M_DO                     := M 3035.0);
      NOP   0;
NETWORK
TITLE = SP, MD, TZ 
      A(;
      ON    "md_ds3";
      O     "sp_ds3";
      );
      A     #bypass;
      R     M 3035.0;
NETWORK
TITLE =
      A     M 3035.0;
      =     "QDS3";
NETWORK
TITLE = ФТ-1 ручное управление
      A     M 2005.2;
      =     L 38.0;
      BLD   103;
      A     M 2015.2;
      =     L 38.1;
      BLD   103;
      A     M 2025.2;
      =     L 38.2;
      BLD   103;
      CALL  "DO_MANUAL" (
           MANUAL                   := L 38.0,
           PUSK                     := L 38.1,
           STOP                     := L 38.2,
           M_DO                     := M 3035.2);
      NOP   0;
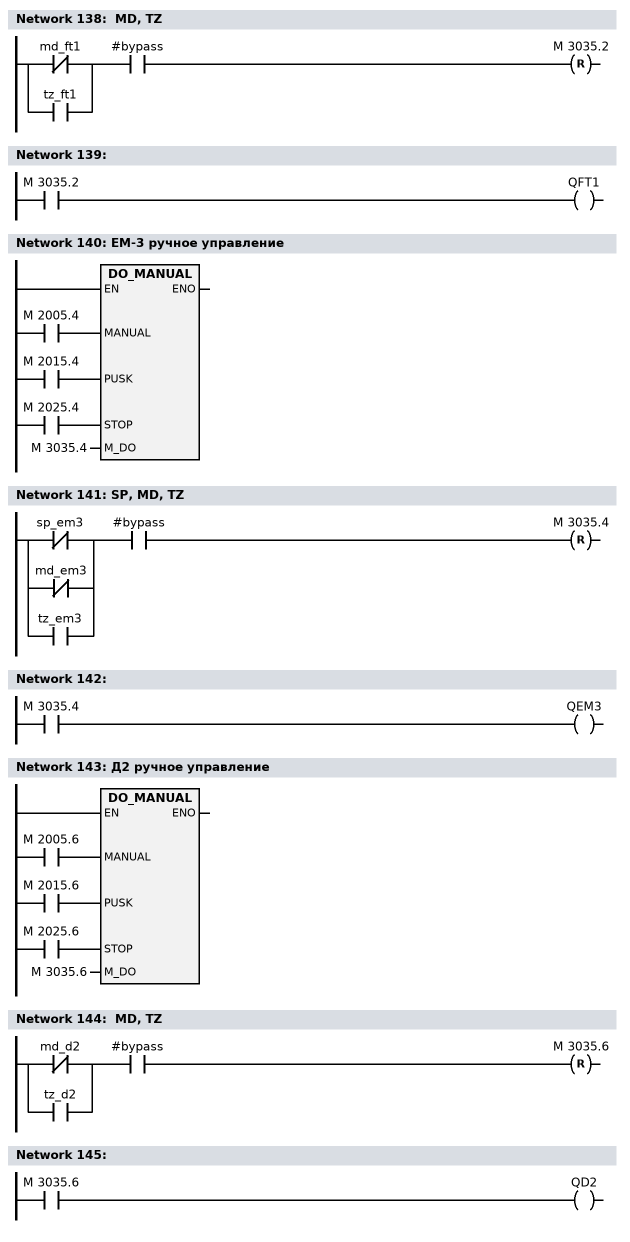
NETWORK
TITLE =  MD, TZ 
      A(;
      ON    "md_ft1";
      O     "tz_ft1";
      );
      A     #bypass;
      R     M 3035.2;
NETWORK
TITLE =
      A     M 3035.2;
      =     "QFT1";
NETWORK
TITLE = ЕМ-3 ручное управление
      A     M 2005.4;
      =     L 38.0;
      BLD   103;
      A     M 2015.4;
      =     L 38.1;
      BLD   103;
      A     M 2025.4;
      =     L 38.2;
      BLD   103;
      CALL  "DO_MANUAL" (
           MANUAL                   := L 38.0,
           PUSK                     := L 38.1,
           STOP                     := L 38.2,
           M_DO                     := M 3035.4);
      NOP   0;
NETWORK
TITLE = SP, MD, TZ 
      A(;
      ON    "sp_em3";
      ON    "md_em3";
      O     "tz_em3";
      );
      A     #bypass;
      R     M 3035.4;
NETWORK
TITLE =
      A     M 3035.4;
      =     "QEM3";
NETWORK
TITLE = Д2 ручное управление
      A     M 2005.6;
      =     L 38.0;
      BLD   103;
      A     M 2015.6;
      =     L 38.1;
      BLD   103;
      A     M 2025.6;
      =     L 38.2;
      BLD   103;
      CALL  "DO_MANUAL" (
           MANUAL                   := L 38.0,
           PUSK                     := L 38.1,
           STOP                     := L 38.2,
           M_DO                     := M 3035.6);
      NOP   0;
NETWORK
TITLE =  MD, TZ 
      A(;
      ON    "md_d2";
      O     "tz_d2";
      );
      A     #bypass;
      R     M 3035.6;
NETWORK
TITLE =
      A     M 3035.6;
      =     "QD2";
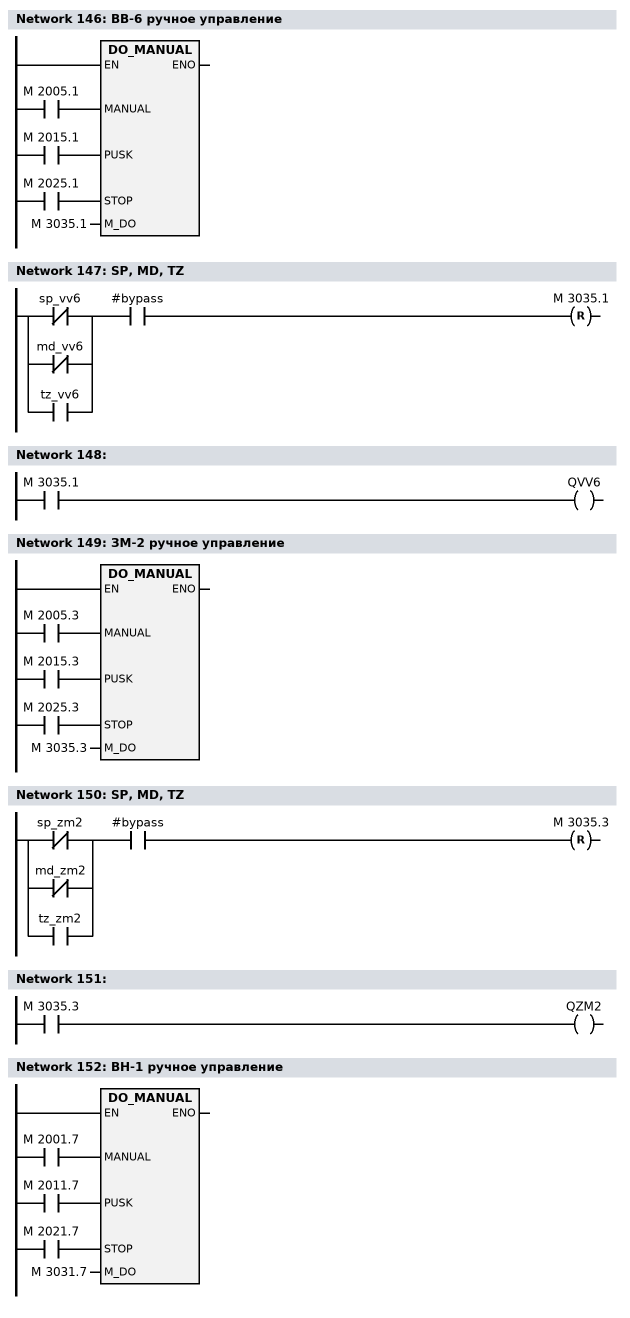
NETWORK
TITLE = ВВ-6 ручное управление
      A     M 2005.1;
      =     L 38.0;
      BLD   103;
      A     M 2015.1;
      =     L 38.1;
      BLD   103;
      A     M 2025.1;
      =     L 38.2;
      BLD   103;
      CALL  "DO_MANUAL" (
           MANUAL                   := L 38.0,
           PUSK                     := L 38.1,
           STOP                     := L 38.2,
           M_DO                     := M 3035.1);
      NOP   0;
NETWORK
TITLE = SP, MD, TZ 
      A(;
      ON    "sp_vv6";
      ON    "md_vv6";
      O     "tz_vv6";
      );
      A     #bypass;
      R     M 3035.1;
NETWORK
TITLE =
      A     M 3035.1;
      =     "QVV6";
NETWORK
TITLE = ЗМ-2 ручное управление
      A     M 2005.3;
      =     L 38.0;
      BLD   103;
      A     M 2015.3;
      =     L 38.1;
      BLD   103;
      A     M 2025.3;
      =     L 38.2;
      BLD   103;
      CALL  "DO_MANUAL" (
           MANUAL                   := L 38.0,
           PUSK                     := L 38.1,
           STOP                     := L 38.2,
           M_DO                     := M 3035.3);
      NOP   0;
NETWORK
TITLE = SP, MD, TZ 
      A(;
      ON    "sp_zm2";
      ON    "md_zm2";
      O     "tz_zm2";
      );
      A     #bypass;
      R     M 3035.3;
NETWORK
TITLE =
      A     M 3035.3;
      =     "QZM2";
NETWORK
TITLE = ВН-1 ручное управление
      A     M 2001.7;
      =     L 38.0;
      BLD   103;
      A     M 2011.7;
      =     L 38.1;
      BLD   103;
      A     M 2021.7;
      =     L 38.2;
      BLD   103;
      CALL  "DO_MANUAL" (
           MANUAL                   := L 38.0,
           PUSK                     := L 38.1,
           STOP                     := L 38.2,
           M_DO                     := M 3031.7);
      NOP   0;
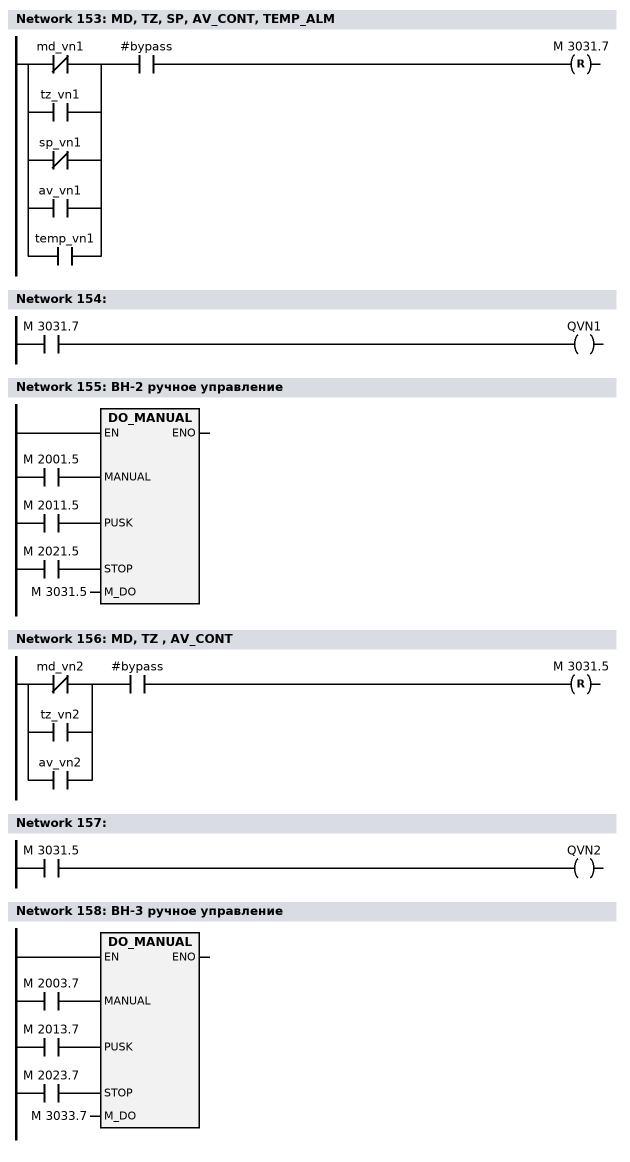
NETWORK
TITLE = MD, TZ, SP, AV_CONT, TEMP_ALM
      A(;
      ON    "md_vn1";
      O     "tz_vn1";
      ON    "sp_vn1";
      O     "av_vn1";
      O     "temp_vn1";
      );
      A     #bypass;
      R     M 3031.7;
NETWORK
TITLE =
      A     M 3031.7;
      =     "QVN1";
NETWORK
TITLE = ВН-2 ручное управление
      A     M 2001.5;
      =     L 38.0;
      BLD   103;
      A     M 2011.5;
      =     L 38.1;
      BLD   103;
      A     M 2021.5;
      =     L 38.2;
      BLD   103;
      CALL  "DO_MANUAL" (
           MANUAL                   := L 38.0,
           PUSK                     := L 38.1,
           STOP                     := L 38.2,
           M_DO                     := M 3031.5);
      NOP   0;
NETWORK
TITLE = MD, TZ , AV_CONT
      A(;
      ON    "md_vn2";
      O     "tz_vn2";
      O     "av_vn2";
      );
      A     #bypass;
      R     M 3031.5;
NETWORK
TITLE =
      A     M 3031.5;
      =     "QVN2";
NETWORK
TITLE = ВН-3 ручное управление
      A     M 2003.7;
      =     L 38.0;
      BLD   103;
      A     M 2013.7;
      =     L 38.1;
      BLD   103;
      A     M 2023.7;
      =     L 38.2;
      BLD   103;
      CALL  "DO_MANUAL" (
           MANUAL                   := L 38.0,
           PUSK                     := L 38.1,
           STOP                     := L 38.2,
           M_DO                     := M 3033.7);
      NOP   0;
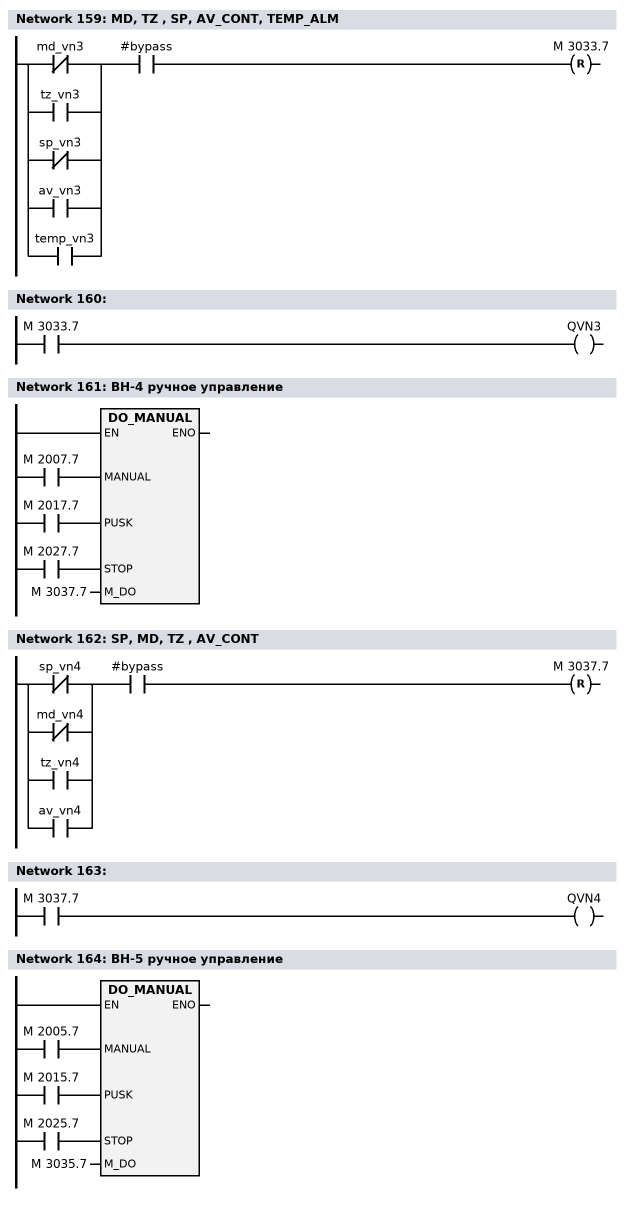
NETWORK
TITLE = MD, TZ , SP, AV_CONT, TEMP_ALM
      A(;
      ON    "md_vn3";
      O     "tz_vn3";
      ON    "sp_vn3";
      O     "av_vn3";
      O     "temp_vn3";
      );
      A     #bypass;
      R     M 3033.7;
NETWORK
TITLE =
      A     M 3033.7;
      =     "QVN3";
NETWORK
TITLE = ВН-4 ручное управление
      A     M 2007.7;
      =     L 38.0;
      BLD   103;
      A     M 2017.7;
      =     L 38.1;
      BLD   103;
      A     M 2027.7;
      =     L 38.2;
      BLD   103;
      CALL  "DO_MANUAL" (
           MANUAL                   := L 38.0,
           PUSK                     := L 38.1,
           STOP                     := L 38.2,
           M_DO                     := M 3037.7);
      NOP   0;
NETWORK
TITLE = SP, MD, TZ , AV_CONT
      A(;
      ON    "sp_vn4";
      ON    "md_vn4";
      O     "tz_vn4";
      O     "av_vn4";
      );
      A     #bypass;
      R     M 3037.7;
NETWORK
TITLE =
      A     M 3037.7;
      =     "QVN4";
NETWORK
TITLE = ВН-5 ручное управление
      A     M 2005.7;
      =     L 38.0;
      BLD   103;
      A     M 2015.7;
      =     L 38.1;
      BLD   103;
      A     M 2025.7;
      =     L 38.2;
      BLD   103;
      CALL  "DO_MANUAL" (
           MANUAL                   := L 38.0,
           PUSK                     := L 38.1,
           STOP                     := L 38.2,
           M_DO                     := M 3035.7);
      NOP   0;
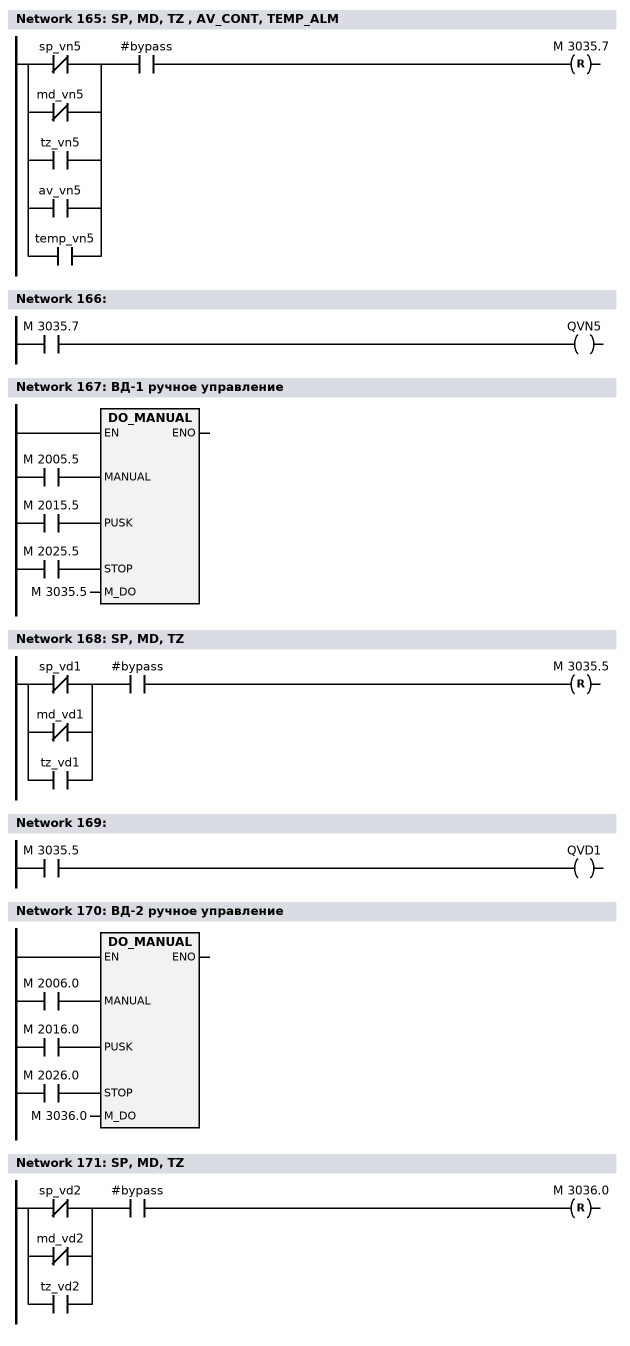
NETWORK
TITLE = SP, MD, TZ , AV_CONT, TEMP_ALM
      A(;
      ON    "sp_vn5";
      ON    "md_vn5";
      O     "tz_vn5";
      O     "av_vn5";
      O     "temp_vn5";
      );
      A     #bypass;
      R     M 3035.7;
NETWORK
TITLE =
      A     M 3035.7;
      =     "QVN5";
NETWORK
TITLE = ВД-1 ручное управление
      A     M 2005.5;
      =     L 38.0;
      BLD   103;
      A     M 2015.5;
      =     L 38.1;
      BLD   103;
      A     M 2025.5;
      =     L 38.2;
      BLD   103;
      CALL  "DO_MANUAL" (
           MANUAL                   := L 38.0,
           PUSK                     := L 38.1,
           STOP                     := L 38.2,
           M_DO                     := M 3035.5);
      NOP   0;
NETWORK
TITLE = SP, MD, TZ 
      A(;
      ON    "sp_vd1";
      ON    "md_vd1";
      O     "tz_vd1";
      );
      A     #bypass;
      R     M 3035.5;
NETWORK
TITLE =
      A     M 3035.5;
      =     "QVD1";
NETWORK
TITLE = ВД-2 ручное управление
      A     M 2006.0;
      =     L 38.0;
      BLD   103;
      A     M 2016.0;
      =     L 38.1;
      BLD   103;
      A     M 2026.0;
      =     L 38.2;
      BLD   103;
      CALL  "DO_MANUAL" (
           MANUAL                   := L 38.0,
           PUSK                     := L 38.1,
           STOP                     := L 38.2,
           M_DO                     := M 3036.0);
      NOP   0;
NETWORK
TITLE = SP, MD, TZ 
      A(;
      ON    "sp_vd2";
      ON    "md_vd2";
      O     "tz_vd2";
      );
      A     #bypass;
      R     M 3036.0;
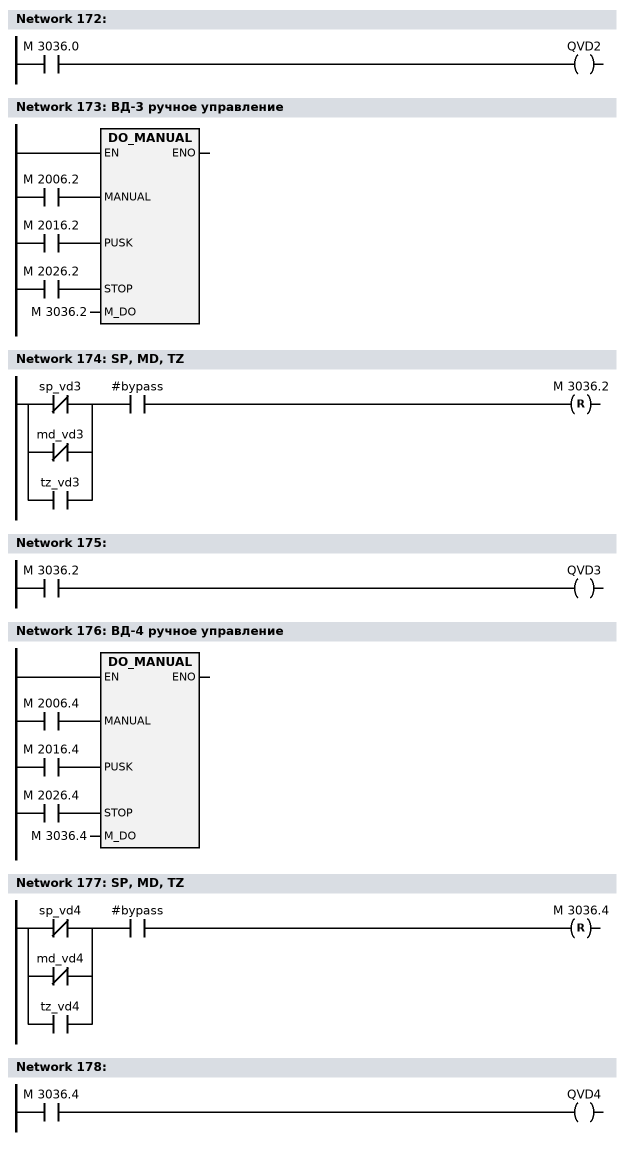
NETWORK
TITLE =
      A     M 3036.0;
      =     "QVD2";
NETWORK
TITLE = ВД-3 ручное управление
      A     M 2006.2;
      =     L 38.0;
      BLD   103;
      A     M 2016.2;
      =     L 38.1;
      BLD   103;
      A     M 2026.2;
      =     L 38.2;
      BLD   103;
      CALL  "DO_MANUAL" (
           MANUAL                   := L 38.0,
           PUSK                     := L 38.1,
           STOP                     := L 38.2,
           M_DO                     := M 3036.2);
      NOP   0;
NETWORK
TITLE = SP, MD, TZ 
      A(;
      ON    "sp_vd3";
      ON    "md_vd3";
      O     "tz_vd3";
      );
      A     #bypass;
      R     M 3036.2;
NETWORK
TITLE =
      A     M 3036.2;
      =     "QVD3";
NETWORK
TITLE = ВД-4 ручное управление
      A     M 2006.4;
      =     L 38.0;
      BLD   103;
      A     M 2016.4;
      =     L 38.1;
      BLD   103;
      A     M 2026.4;
      =     L 38.2;
      BLD   103;
      CALL  "DO_MANUAL" (
           MANUAL                   := L 38.0,
           PUSK                     := L 38.1,
           STOP                     := L 38.2,
           M_DO                     := M 3036.4);
      NOP   0;
NETWORK
TITLE = SP, MD, TZ 
      A(;
      ON    "sp_vd4";
      ON    "md_vd4";
      O     "tz_vd4";
      );
      A     #bypass;
      R     M 3036.4;
NETWORK
TITLE =
      A     M 3036.4;
      =     "QVD4";
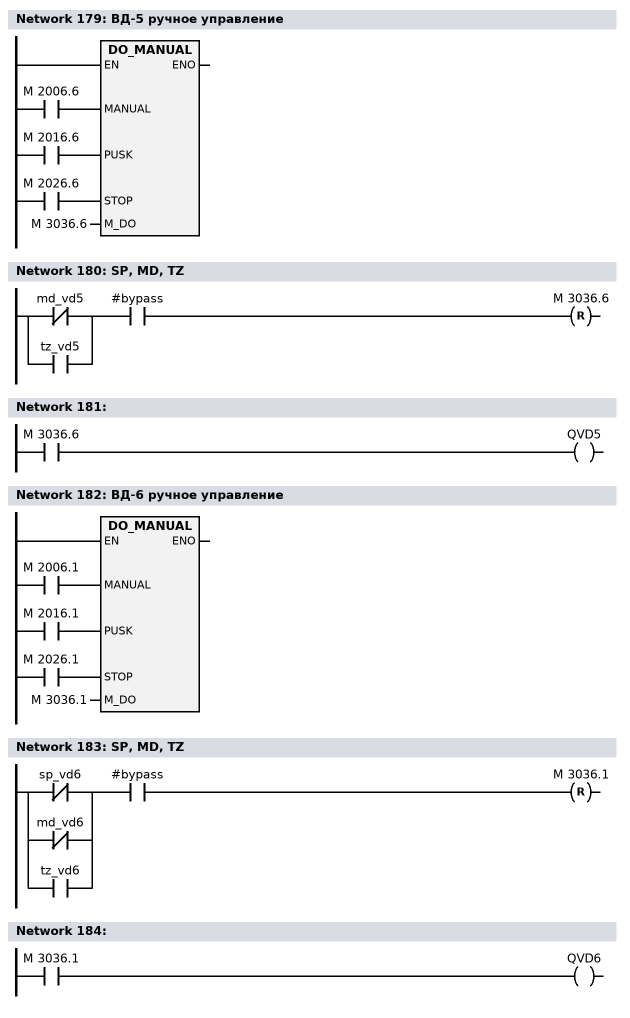
NETWORK
TITLE = ВД-5 ручное управление
      A     M 2006.6;
      =     L 38.0;
      BLD   103;
      A     M 2016.6;
      =     L 38.1;
      BLD   103;
      A     M 2026.6;
      =     L 38.2;
      BLD   103;
      CALL  "DO_MANUAL" (
           MANUAL                   := L 38.0,
           PUSK                     := L 38.1,
           STOP                     := L 38.2,
           M_DO                     := M 3036.6);
      NOP   0;
NETWORK
TITLE = SP, MD, TZ 
      A(;
      ON    "md_vd5";
      O     "tz_vd5";
      );
      A     #bypass;
      R     M 3036.6;
NETWORK
TITLE =
      A     M 3036.6;
      =     "QVD5";
NETWORK
TITLE = ВД-6 ручное управление
      A     M 2006.1;
      =     L 38.0;
      BLD   103;
      A     M 2016.1;
      =     L 38.1;
      BLD   103;
      A     M 2026.1;
      =     L 38.2;
      BLD   103;
      CALL  "DO_MANUAL" (
           MANUAL                   := L 38.0,
           PUSK                     := L 38.1,
           STOP                     := L 38.2,
           M_DO                     := M 3036.1);
      NOP   0;
NETWORK
TITLE = SP, MD, TZ 
      A(;
      ON    "sp_vd6";
      ON    "md_vd6";
      O     "tz_vd6";
      );
      A     #bypass;
      R     M 3036.1;
NETWORK
TITLE =
      A     M 3036.1;
      =     "QVD6";
END_ORGANIZATION_BLOCK
